# EPICS autosave request: softGlueApp/Db/triggerAction_settings.req
$(P)$(Q)softGlueInstance
$(P)$(Q)fieldIOSigNum
$(P)$(Q)trigSseq.LNK1
